{attribute 'GeneratedUsingTerminal: ELX9560-0000-0016'}
{attribute addProperty BoxType "ELX9560-0000-0016"}
{attribute addProperty Id "EtcSlaveTerminalBaseStatus_UinAT %I*Status_Uin_449D6AB51Status_UexAT %I*Status_Uex_449D6AB51WcStateAT %I*WcState_9091E0EB2InfoDataAT %I*InfoData_6F19DB2B2"}
{attribute addProperty CRC "3125350503"}
{attribute addProperty Size "6"}
TYPE ELX9560_BA491067 EXTENDS EtcSlaveTerminalBase :
STRUCT
	{attribute addProperty Name "Status_Uin"}
	Status_Uin : Status_Uin_449D6AB5;
	{attribute addProperty Name "Status_Uex"}
	Status_Uex : Status_Uex_449D6AB5;
	{attribute addProperty Name "WcState"}
	WcState : WcState_9091E0EB;
	{attribute addProperty Name "InfoData"}
	InfoData : InfoData_6F19DB2B;
END_STRUCT
END_TYPE

(* stored: Version 1.2.0.0, ProductVersion 3.1.4024.9
   DUT ELX9560_BA491067: Id {ab1b42d8-1756-4efb-8672-a567e1e73ffc} *)
